FUNCTION_BLOCK FB_DEV_AnaIn EXTENDS FB_DeviceBase IMPLEMENTS ITF_DEV_AnaIn
VAR_INPUT
END_VAR
VAR_OUTPUT
END_VAR
VAR
END_VAR

END_FUNCTION_BLOCK

(* stored: Version 1.1.0.1, ProductVersion 3.1.4024.12
   POU FB_DEV_AnaIn: Id {0af2c6ce-90b5-4234-ac96-b088e81680e4}, SpecialFunc None *)
